// TIA Portal V19 export
FUNCTION_BLOCK "faceplate"   // FB1, LAD
{ S7_Optimized_Access := 'TRUE' }
// stored: MemoryReserve 100, SetENOAutomatically false
   VAR_INPUT
      start : Bool;
      stop : Bool;
   END_VAR
   VAR_OUTPUT
      "conveyor-right" : Bool;
      "conveyor-left" : Bool;
   END_VAR
   VAR_IN_OUT
      "Time-Right" : Time;
      "Time-Right-Rest" : Time;
      "Time-Left" : Time;
      "memory-stop" : Bool;
      "memory-start" : Bool;
      "Time-Left-Rest" : Time;
   END_VAR
   VAR
      "Timer-Right" : TP_TIME;
      "Timer-Right-Rest" : TP_TIME;
      "Timer-Left" : TP_TIME;
      "Timer-Left-Rest" : TP_TIME;
      "mem-start" : Bool;
      "mem-stop" : Bool;
      "mem-edge-1" : Bool;
      "mem-edge-2" : Bool;
      "mem-edge-3" : Bool;
      "mem-edge-4" : Bool;
      "mem-edge-5" : Bool;
      "mem-edge-6" : Bool;
   END_VAR
   VAR_TEMP   // added for the SCL form of the ladder/FBD networks
      _w1 : Bool;
   END_VAR
BEGIN

REGION Network 1
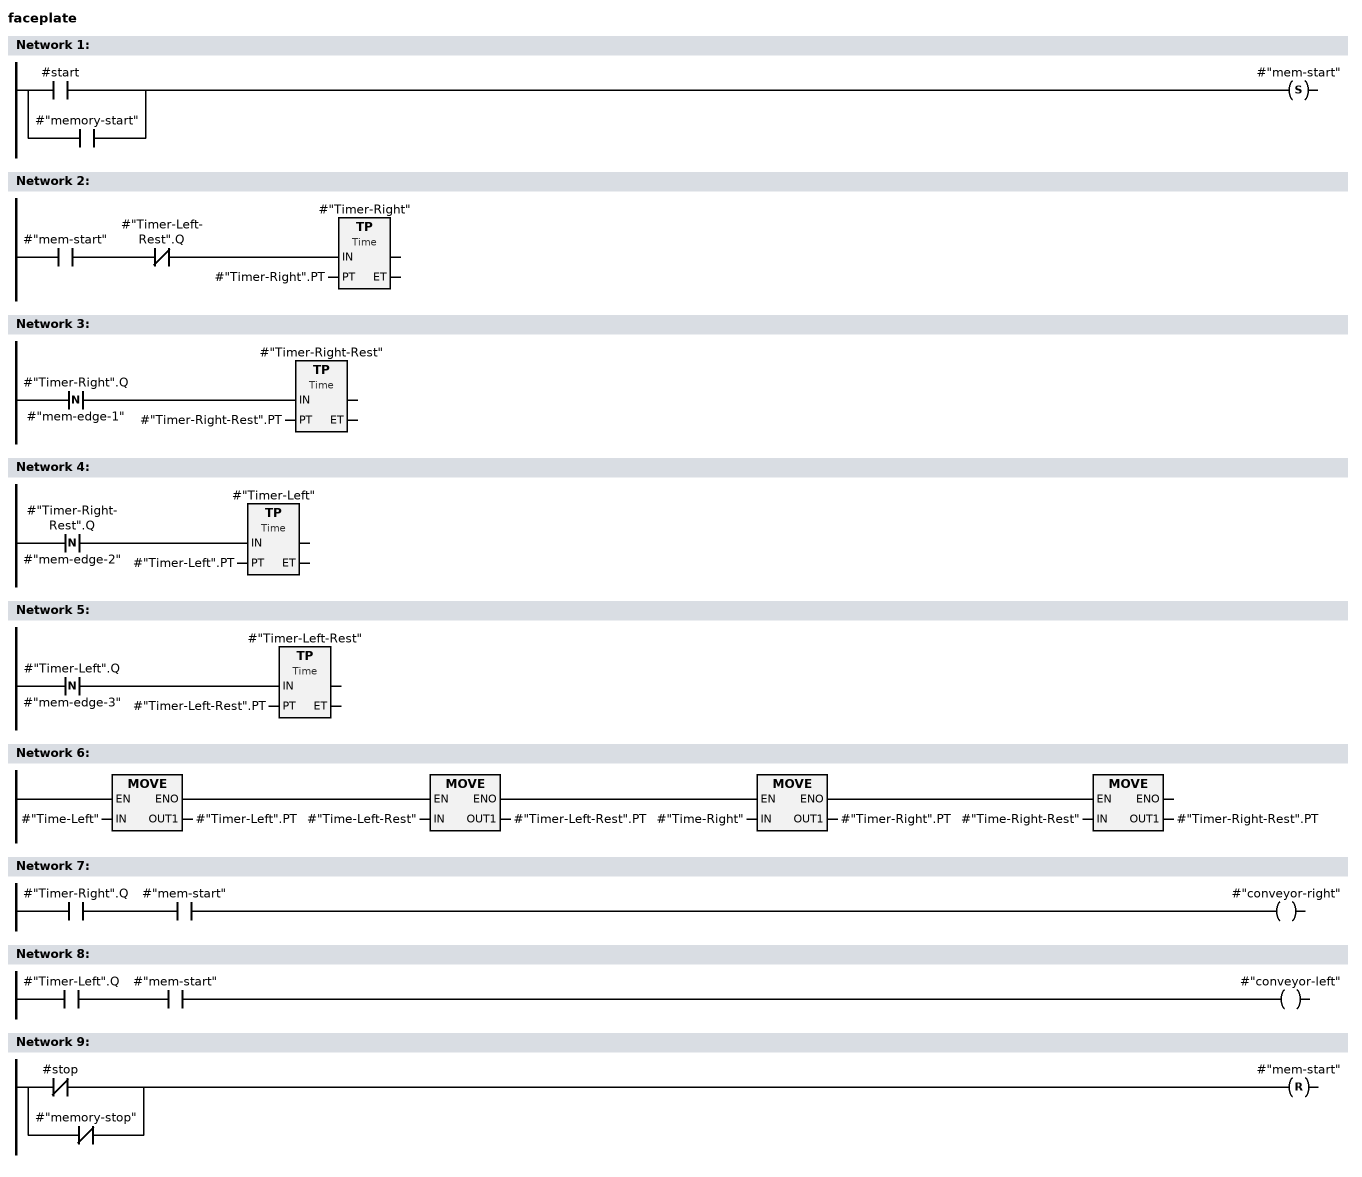
   RUNG wire#powerrail
      Contact( #start )
      wire#w1
      S_Coil( #"mem-start" )
   END_RUNG
   RUNG wire#powerrail
      Contact( #"memory-start" )
   END_RUNG wire#w1
   // the same network as SCL:
   IF #start OR #"memory-start" THEN #"mem-start" := TRUE; END_IF;
END_REGION

REGION Network 2
   RUNG wire#powerrail
      Contact( #"mem-start" )
      I_Contact( #"Timer-Left-Rest".Q )
      { S7_Templates := "time_type := Time" } #"Timer-Right".TP(pt := #"Timer-Right".PT, et =>)
   END_RUNG
   // the same network as SCL:
   #"Timer-Right"(IN := #"mem-start" AND NOT #"Timer-Left-Rest".Q, PT := #"Timer-Right".PT);   // TP
END_REGION

REGION Network 3
   RUNG wire#powerrail
      N_Contact(operand := #"Timer-Right".Q, bit := #"mem-edge-1")
      { S7_Templates := "time_type := Time" } #"Timer-Right-Rest".TP(pt := #"Timer-Right-Rest".PT, et =>)
   END_RUNG
   // the same network as SCL:
   #_w1 := NOT #"Timer-Right".Q AND #"mem-edge-1";   // falling edge of #"Timer-Right".Q
   #"mem-edge-1" := #"Timer-Right".Q;
   #"Timer-Right-Rest"(IN := #_w1, PT := #"Timer-Right-Rest".PT);   // TP
END_REGION

REGION Network 4
   RUNG wire#powerrail
      N_Contact(operand := #"Timer-Right-Rest".Q, bit := #"mem-edge-2")
      { S7_Templates := "time_type := Time" } #"Timer-Left".TP(pt := #"Timer-Left".PT, et =>)
   END_RUNG
   // the same network as SCL:
   #_w1 := NOT #"Timer-Right-Rest".Q AND #"mem-edge-2";   // falling edge of #"Timer-Right-Rest".Q
   #"mem-edge-2" := #"Timer-Right-Rest".Q;
   #"Timer-Left"(IN := #_w1, PT := #"Timer-Left".PT);   // TP
END_REGION

REGION Network 5
   RUNG wire#powerrail
      N_Contact(operand := #"Timer-Left".Q, bit := #"mem-edge-3")
      { S7_Templates := "time_type := Time" } #"Timer-Left-Rest".TP(pt := #"Timer-Left-Rest".PT, et =>)
   END_RUNG
   // the same network as SCL:
   #_w1 := NOT #"Timer-Left".Q AND #"mem-edge-3";   // falling edge of #"Timer-Left".Q
   #"mem-edge-3" := #"Timer-Left".Q;
   #"Timer-Left-Rest"(IN := #_w1, PT := #"Timer-Left-Rest".PT);   // TP
END_REGION

REGION Network 6
   RUNG wire#powerrail
      Move(in := #"Time-Left", out1 => #"Timer-Left".PT)
      Move(in := #"Time-Left-Rest", out1 => #"Timer-Left-Rest".PT)
      Move(in := #"Time-Right", out1 => #"Timer-Right".PT)
      Move(in := #"Time-Right-Rest", out1 => #"Timer-Right-Rest".PT)
   END_RUNG
   // the same network as SCL:
   #"Timer-Left".PT := #"Time-Left";
   #"Timer-Left-Rest".PT := #"Time-Left-Rest";
   #"Timer-Right".PT := #"Time-Right";
   #"Timer-Right-Rest".PT := #"Time-Right-Rest";
END_REGION

REGION Network 7
   RUNG wire#powerrail
      Contact( #"Timer-Right".Q )
      Contact( #"mem-start" )
      Coil( #"conveyor-right" )
   END_RUNG
   // the same network as SCL:
   #"conveyor-right" := #"Timer-Right".Q AND #"mem-start";
END_REGION

REGION Network 8
   RUNG wire#powerrail
      Contact( #"Timer-Left".Q )
      Contact( #"mem-start" )
      Coil( #"conveyor-left" )
   END_RUNG
   // the same network as SCL:
   #"conveyor-left" := #"Timer-Left".Q AND #"mem-start";
END_REGION

REGION Network 9
   RUNG wire#powerrail
      I_Contact( #stop )
      wire#w1
      R_Coil( #"mem-start" )
   END_RUNG
   RUNG wire#powerrail
      I_Contact( #"memory-stop" )
   END_RUNG wire#w1
   // the same network as SCL:
   IF NOT #stop OR NOT #"memory-stop" THEN #"mem-start" := FALSE; END_IF;
END_REGION
END_FUNCTION_BLOCK
